FUNCTION_BLOCK FB_Regelschuif_DG IMPLEMENTS ITF_Regelschuif
VAR
	TagName: STRING;
	
	OpenSchuif: ITF_Regelschuif_OutOpen_DG;
	SluitSchuif: ITF_Regelschuif_OutClose_DG;
	InputSchuif: ITF_Regelschuif_In_DG;
	
	CurrentMode: E_Bedrijfstoestand:= E_Bedrijfstoestand.off;
	
	SchuifPosition: SINT;
	VorigePosition: SINT;
	Marge : SINT := 2;
	
	error_Trigger: R_TRIG;
	ErrorTimer: TON;
END_VAR

//De errortimer wordt gestart zodra de schuif niet in standby staat en de timer niet is afgelopen
ErrorTimer(IN:= StateRegelschuif <> E_Regelschuifstate.standby AND NOT ErrorTimer.Q ,PT:= T#5S);

//Als de schuif uit staat stopt de regelschuif met openen of sluiten
IF CurrentMode = E_Bedrijfstoestand.off THEN
	Openschuif.set(FALSE);
	SluitSchuif.set(FALSE);
END_IF

//De actuele positie van de schuif wordt opgehaald
ActueelPosition:= InputSchuif.get();
SchuifPosition:= InputSchuif.get();

error_Trigger(CLK:= ErrorTimer.Q);

IF error_Trigger.Q THEN
	IF (ActueelPosition < (Vorigeposition + Marge) AND StateRegelschuif = E_Regelschuifstate.opening) OR
		(ActueelPosition > (Vorigeposition - Marge) AND StateRegelschuif = E_Regelschuifstate.closing)THEN
		Stateregelschuif:= E_RegelschuifState.error;
		main.alarms.Append(tag:= TagName, msg := 'Schuifstroing gedetecteerd: Schuif beweegt niet binnen de marge');
	END_IF
	VorigePosition := ActueelPosition;
END_IF

IF (ActueelPosition > (Vorigeposition + Marge) AND Stateregelschuif = E_RegelschuifState.error) THEN
Stateregelschuif := E_RegelschuifState.opening;
END_IF

PROPERTY ActueelPosition : SINT
GET
END_GET
SET
END_SET
END_PROPERTY

METHOD FB_init : BOOL
VAR_INPUT
	bInitRetains : BOOL; // if TRUE, the retain variables are initialized (warm start / cold start)
	bInCopyCode : BOOL;  // if TRUE, the instance afterwards gets moved into the copy code (online change)
	
	tag: STRING;
	SchuifInput: ITF_Regelschuif_In_DG;
	OutputOpen: ITF_Regelschuif_OutOpen_DG;
	OutputClose: ITF_Regelschuif_OutClose_DG;
	
END_VAR
TagName:= tag;
InputSchuif := SchuifInput;
OpenSchuif := OutputOpen;
SluitSchuif := OutputClose;
END_METHOD

METHOD RegelSchuifGoTo : SINT
VAR
	PulseTimer: TON;
	StartPulse: BOOL := TRUE;
	OpenTimer: TON;
	StartOpen: BOOL := FALSE;
END_VAR
VAR_INPUT
	regelschuifdoel: SINT;
END_VAR
//Zet de timer voor de puls op 1 minuut/10 seconden voor testen
PulseTimer(IN:=StartPulse ,PT:= T#10S);
Opentimer(IN:=StartOpen , PT:= T#1S);

regelschuifdoel := Inputschuif.get();

IF PulseTimer.Q AND (stateRegelschuif <> E_RegelschuifState.error) AND (Currentmode <> E_Bedrijfstoestand.off) THEN
	//Als de regelschuif zijn actuele positie op zijn doel is wordt hij uitgezet
	IF (regelschuifdoel = ActueelPosition)THEN
		StateRegelschuif := E_RegelschuifState.standby;
	END_IF
	//Als het doel kleiner is dan de actuele positie gaat hij sluiten
	IF (regelschuifdoel < ActueelPosition) THEN
		StateRegelschuif := E_RegelschuifState.closing;
		OpenSchuif.set(FALSE);
		SluitSchuif.set(TRUE);
	END_IF
	//Als het doel groter is dan de actuele positie gaat hij openen
	IF (regelschuifdoel > ActueelPosition) THEN
		StateRegelschuif := E_RegelschuifState.opening;
		OpenSchuif.set(TRUE);
		Sluitschuif.set(FALSE);
	END_IF	
	StartPulse := FALSE;
	StartPulse := TRUE;
END_IF 	

//De regelschuif wordt geopend
IF StateRegelschuif = E_RegelschuifState.opening THEN
	StartOpen := TRUE;
	IF OpenTimer.Q THEN
	ActueelPosition := ActueelPosition + 1;
	END_IF
	StartOpen := FALSE;
END_IF

//De regelschuif wordt gesloten
IF StateRegelschuif = E_RegelschuifState.closing THEN
	StartOpen := TRUE;
	IF OpenTimer.Q THEN
	ActueelPosition := ActueelPosition - 1;
	END_IF
	StartOpen := FALSE;
END_IF

//Zorgt ervoor dat de schuif stopt met bewegen als hij wordt uitgeschakeld
IF CurrentMode = E_Bedrijfstoestand.off THEN
	regelschuifdoel := ActueelPosition;
END_IF
END_METHOD

PROPERTY StateRegelschuif : E_RegelschuifState
GET
END_GET
SET
END_SET
END_PROPERTY

END_FUNCTION_BLOCK

(* stored: Version 1.1.0.1, ProductVersion 3.1.4026.8
   POU FB_Regelschuif_DG: Id {197a057b-7e77-4001-97d3-497a9b935830}, SpecialFunc None
   Folder Methods: Id {a5c8f5f8-d7b2-406e-83cb-5c27f5fd8301}
   Folder Properties: Id {b6eb3f6c-3011-4a7e-8816-c7f569303f45}
   Property ActueelPosition: Id {e5264e59-d7b3-4d52-85a9-01c31af68424}
   Get Get: Id {9fd5639f-907b-4f81-9ddb-25b621dd3e75}
   Set Set: Id {905c9011-2b5d-48ef-959c-c4e2af0ee1b8}
   Method FB_init: Id {f3ca1436-908a-411d-9d51-011caa116cfc}
   Method RegelschuifGoTo: Id {a4a1d9ca-2482-46aa-ba66-9fb460cea5bb}
   Property StateRegelschuif: Id {6308ac59-5f2f-4aa8-a02c-ba74a875ce56}
   Get Get: Id {9fed2dd4-a8a2-4e9a-a768-d82a5581c148}
   Set Set: Id {39e89b3f-9284-4275-8393-d34cd7d64bd6} *)
